// Mitsubishi GX Works2 project: servo_Mcode_0911   PLC: Q02/Q02H

PROGRAM MAIN
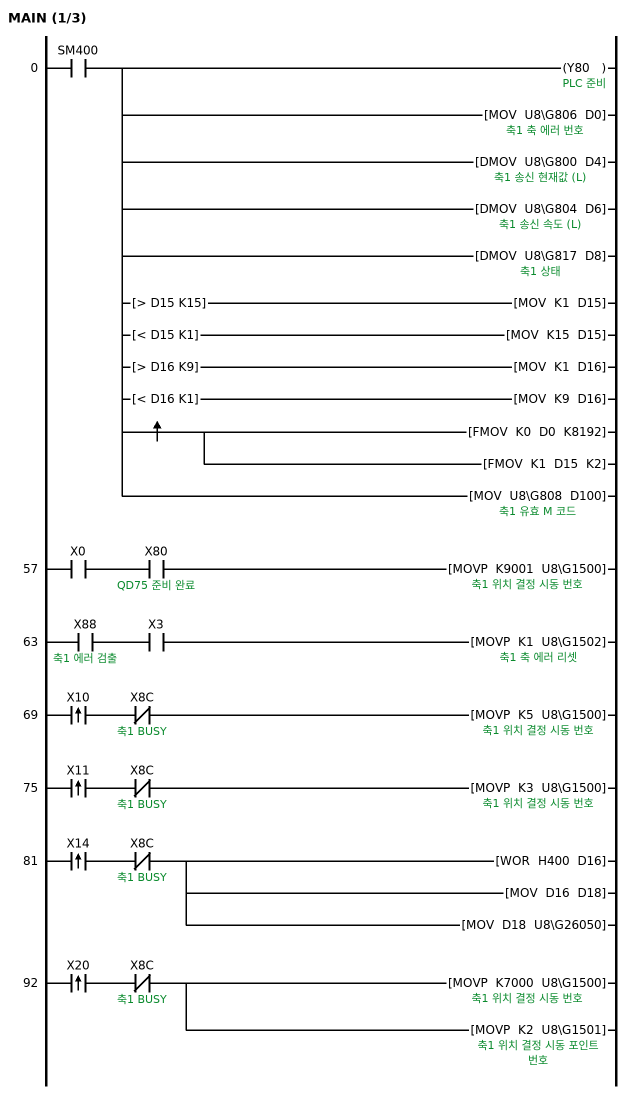
0     LD      SM400
      OUT     Y80  ; PLC 준비
      MOV     U8\G806 D0  ; 축1 축 에러 번호
      DMOV    U8\G800 D4  ; 축1 송신 현재값 (L)
      DMOV    U8\G804 D6  ; 축1 송신 속도 (L)
      DMOV    U8\G817 D8  ; 축1 상태
      MPS
      AND>    D15 K15
      MOV     K1 D15
      MRD
      AND<    D15 K1
      MOV     K15 D15
      MRD
      AND>    D16 K9
      MOV     K1 D16
      MRD
      AND<    D16 K1
      MOV     K9 D16
      MRD
      MEP
      FMOV    K0 D0 K8192
      FMOV    K1 D15 K2
      MPP
      MOV     U8\G808 D100  ; 축1 유효 M 코드
57    LD      X0
      AND     X80  ; QD75 준비 완료
      MOVP    K9001 U8\G1500  ; 축1 위치 결정 시동 번호
63    LD      X88  ; 축1 에러 검출
      AND     X3
      MOVP    K1 U8\G1502  ; 축1 축 에러 리셋
69    LDP     X10
      ANI     X8C  ; 축1 BUSY
      MOVP    K5 U8\G1500
75    LDP     X11
      ANI     X8C  ; 축1 BUSY
      MOVP    K3 U8\G1500
81    LDP     X14
      ANI     X8C  ; 축1 BUSY
      WOR     H400 D16
      MOV     D16 D18
      MOV     D18 U8\G26050
92    LDP     X20
      ANI     X8C  ; 축1 BUSY
      MOVP    K7000 U8\G1500
      MOVP    K2 U8\G1501  ; 축1 위치 결정 시동 포인트 번호
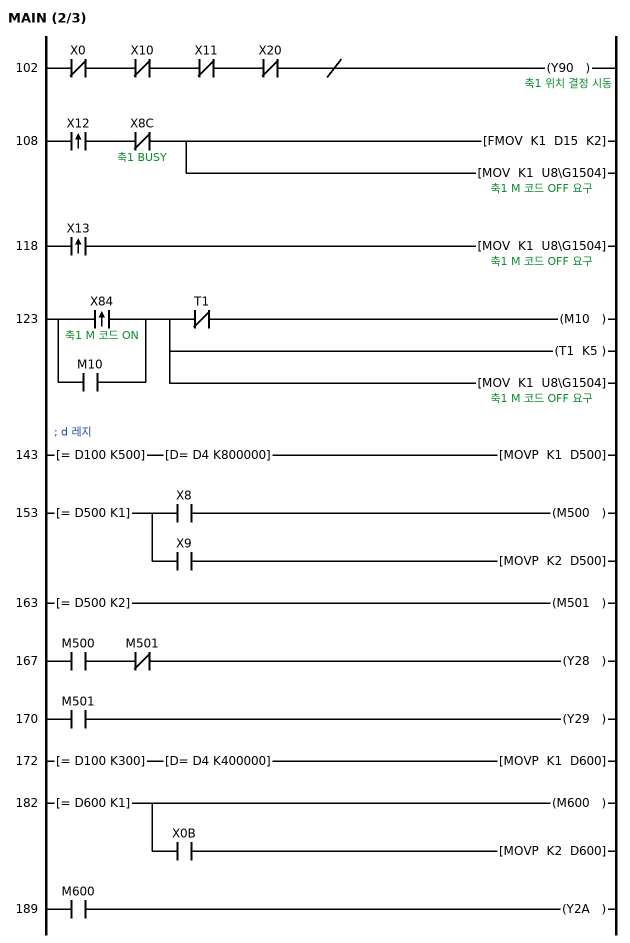
102   LDI     X0
      ANI     X10
      ANI     X11
      ANI     X20
      INV
      OUT     Y90  ; 축1 위치 결정 시동
108   LDP     X12
      ANI     X8C  ; 축1 BUSY
      FMOV    K1 D15 K2
      MOV     K1 U8\G1504  ; 축1 M 코드 OFF 요구
118   LDP     X13
      MOV     K1 U8\G1504
123   LDP     X84  ; 축1 M 코드 ON
      OR      M10
      MPS
      ANI     T1
      OUT     M10
      MPP
      OUT     T1 K5
      MOV     K1 U8\G1504
; d 레지
143   LD=     D100 K500
      ANDD=   D4 K800000
      MOVP    K1 D500
153   LD=     D500 K1
      MPS
      AND     X8
      OUT     M500
      MPP
      AND     X9
      MOVP    K2 D500
163   LD=     D500 K2
      OUT     M501
167   LD      M500
      ANI     M501
      OUT     Y28
170   LD      M501
      OUT     Y29
172   LD=     D100 K300
      ANDD=   D4 K400000
      MOVP    K1 D600
182   LD=     D600 K1
      OUT     M600
      AND     X0B
      MOVP    K2 D600
189   LD      M600
      OUT     Y2A
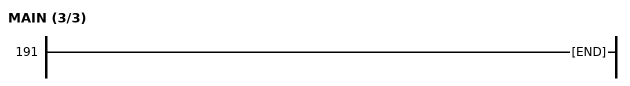
191   END
END_PROGRAM

PROGRAM MAIN1
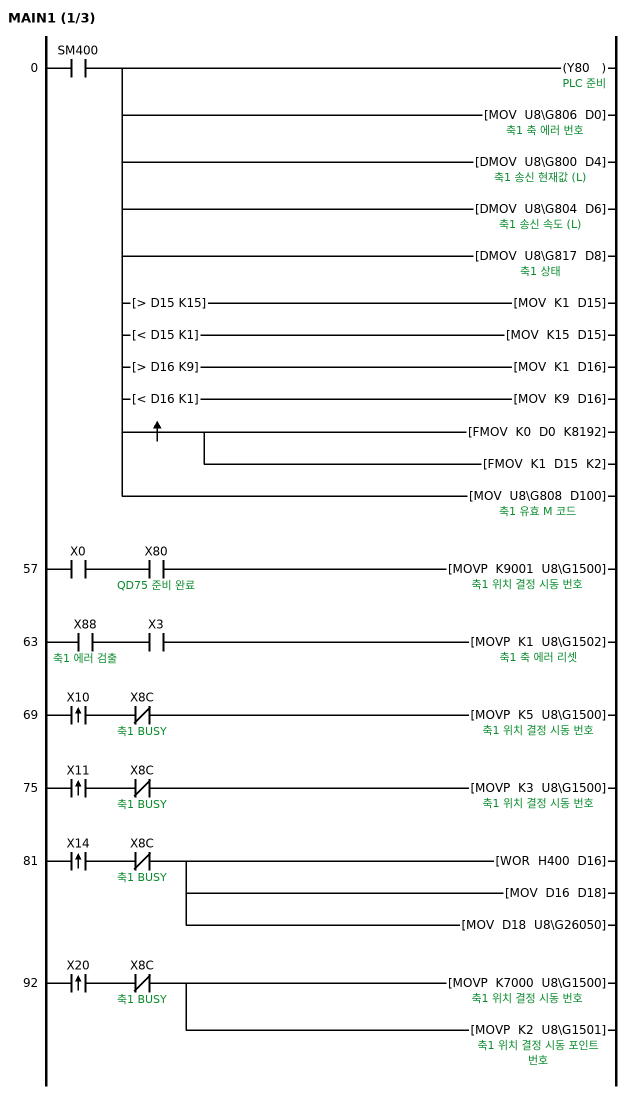
0     LD      SM400
      OUT     Y80  ; PLC 준비
      MOV     U8\G806 D0  ; 축1 축 에러 번호
      DMOV    U8\G800 D4  ; 축1 송신 현재값 (L)
      DMOV    U8\G804 D6  ; 축1 송신 속도 (L)
      DMOV    U8\G817 D8  ; 축1 상태
      MPS
      AND>    D15 K15
      MOV     K1 D15
      MRD
      AND<    D15 K1
      MOV     K15 D15
      MRD
      AND>    D16 K9
      MOV     K1 D16
      MRD
      AND<    D16 K1
      MOV     K9 D16
      MRD
      MEP
      FMOV    K0 D0 K8192
      FMOV    K1 D15 K2
      MPP
      MOV     U8\G808 D100  ; 축1 유효 M 코드
57    LD      X0
      AND     X80  ; QD75 준비 완료
      MOVP    K9001 U8\G1500  ; 축1 위치 결정 시동 번호
63    LD      X88  ; 축1 에러 검출
      AND     X3
      MOVP    K1 U8\G1502  ; 축1 축 에러 리셋
69    LDP     X10
      ANI     X8C  ; 축1 BUSY
      MOVP    K5 U8\G1500
75    LDP     X11
      ANI     X8C  ; 축1 BUSY
      MOVP    K3 U8\G1500
81    LDP     X14
      ANI     X8C  ; 축1 BUSY
      WOR     H400 D16
      MOV     D16 D18
      MOV     D18 U8\G26050
92    LDP     X20
      ANI     X8C  ; 축1 BUSY
      MOVP    K7000 U8\G1500
      MOVP    K2 U8\G1501  ; 축1 위치 결정 시동 포인트 번호
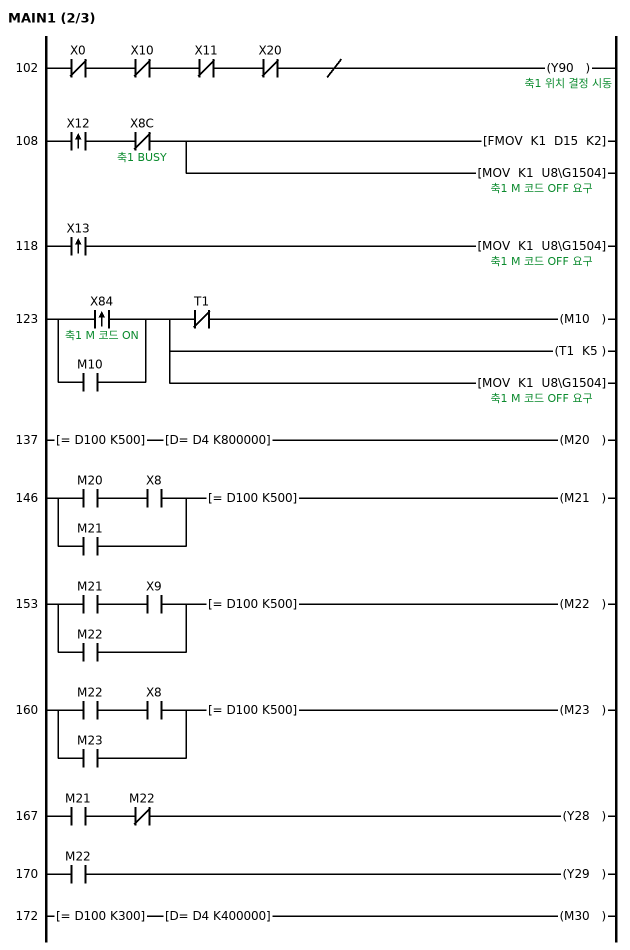
102   LDI     X0
      ANI     X10
      ANI     X11
      ANI     X20
      INV
      OUT     Y90  ; 축1 위치 결정 시동
108   LDP     X12
      ANI     X8C  ; 축1 BUSY
      FMOV    K1 D15 K2
      MOV     K1 U8\G1504  ; 축1 M 코드 OFF 요구
118   LDP     X13
      MOV     K1 U8\G1504
123   LDP     X84  ; 축1 M 코드 ON
      OR      M10
      MPS
      ANI     T1
      OUT     M10
      MPP
      OUT     T1 K5
      MOV     K1 U8\G1504
137   LD=     D100 K500
      ANDD=   D4 K800000
      OUT     M20
146   LD      M20
      AND     X8
      OR      M21
      AND=    D100 K500
      OUT     M21
153   LD      M21
      AND     X9
      OR      M22
      AND=    D100 K500
      OUT     M22
160   LD      M22
      AND     X8
      OR      M23
      AND=    D100 K500
      OUT     M23
167   LD      M21
      ANI     M22
      OUT     Y28
170   LD      M22
      OUT     Y29
172   LD=     D100 K300
      ANDD=   D4 K400000
      OUT     M30
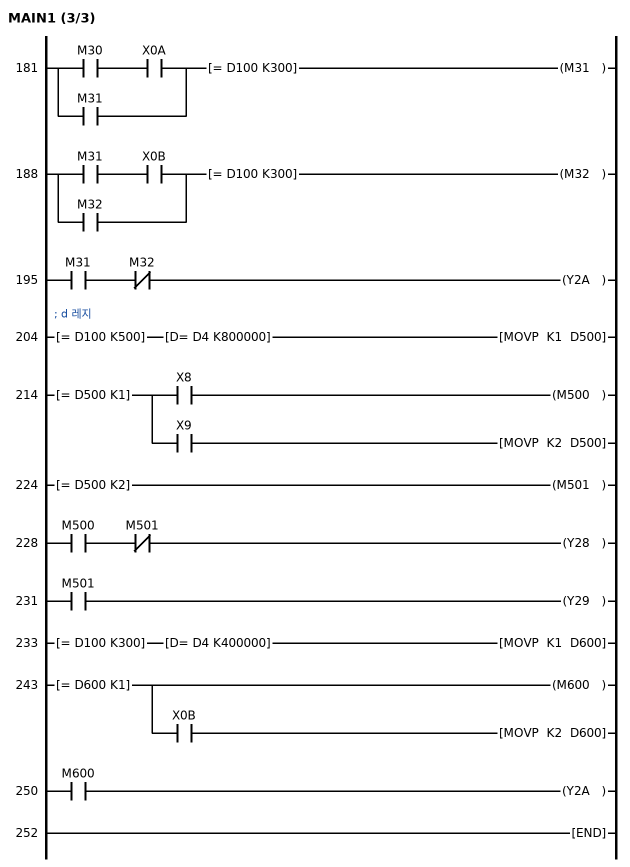
181   LD      M30
      AND     X0A
      OR      M31
      AND=    D100 K300
      OUT     M31
188   LD      M31
      AND     X0B
      OR      M32
      AND=    D100 K300
      OUT     M32
195   LD      M31
      ANI     M32
      OUT     Y2A
; d 레지
204   LD=     D100 K500
      ANDD=   D4 K800000
      MOVP    K1 D500
214   LD=     D500 K1
      MPS
      AND     X8
      OUT     M500
      MPP
      AND     X9
      MOVP    K2 D500
224   LD=     D500 K2
      OUT     M501
228   LD      M500
      ANI     M501
      OUT     Y28
231   LD      M501
      OUT     Y29
233   LD=     D100 K300
      ANDD=   D4 K400000
      MOVP    K1 D600
243   LD=     D600 K1
      OUT     M600
      AND     X0B
      MOVP    K2 D600
250   LD      M600
      OUT     Y2A
252   END
END_PROGRAM

// device comments not shown above
X81  ; 동기용 플래그
X85  ; 축2 M 코드 ON
X89  ; 축2 에러 검출
X8D  ; 축2 BUSY
X90  ; 축1 시동 완료
X91  ; 축2 시동 완료
X94  ; 축1 위치 결정 완료
X95  ; 축2 위치 결정 완료
Y84  ; 축1 축 정지
Y85  ; 축2 축 정지
Y88  ; 축1 정운전 JOG 시동
Y89  ; 축1 역운전 JOG 시동
Y8A  ; 축2 정운전 JOG 시동
Y8B  ; 축2 역운전 JOG 시동
Y91  ; 축2 위치 결정 시동
Y94  ; 축1 실행 금지 플래그
Y95  ; 축2 실행 금지 플래그
